{attribute 'GeneratedUsingTerminal: EK1100-0000-0018'}
{attribute addProperty BoxType "EK1100-0000-0018"}
{attribute addProperty Id "Beckhoff_ER1xxxEK1122Beckhoff_ER1xxxEK1122_892D4B6E492"}
{attribute addProperty CRC "669997616"}
{attribute addProperty Size "492"}
TYPE Beckhoff_ER1xxx_27EF5A30 EXTENDS EK1100_1FC0878B :
STRUCT
	{attribute addProperty Name "Beckhoff_ER1xxxEK1122"}
	{attribute addProperty PreviousPort "Beckhoff ER1xxx : B"}
	Beckhoff_ER1xxxEK1122 : Beckhoff_ER1xxxEK1122_892D4B6E;
END_STRUCT
END_TYPE

(* stored: Version 1.2.0.0, ProductVersion 3.1.4024.9
   DUT Beckhoff_ER1xxx_27EF5A30: Id {4ddcdbc5-13f7-49f3-bf55-09948def3b1f} *)
